FUNCTION_BLOCK SawmillMessageHandler
  (* Standard: 61499-2 *)
  (* Version 0.1, 2017-00-16, hpea485, UOA *)
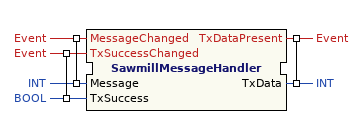
  EVENT_INPUT
    MessageChanged WITH Message;
    TxSuccessChanged WITH TxSuccess;
  END_EVENT
  EVENT_OUTPUT
    TxDataPresent WITH TxData;
  END_EVENT
  VAR_INPUT
    Message : INT;
    TxSuccess : BOOL;
  END_VAR
  VAR_OUTPUT
    TxData : INT;
  END_VAR
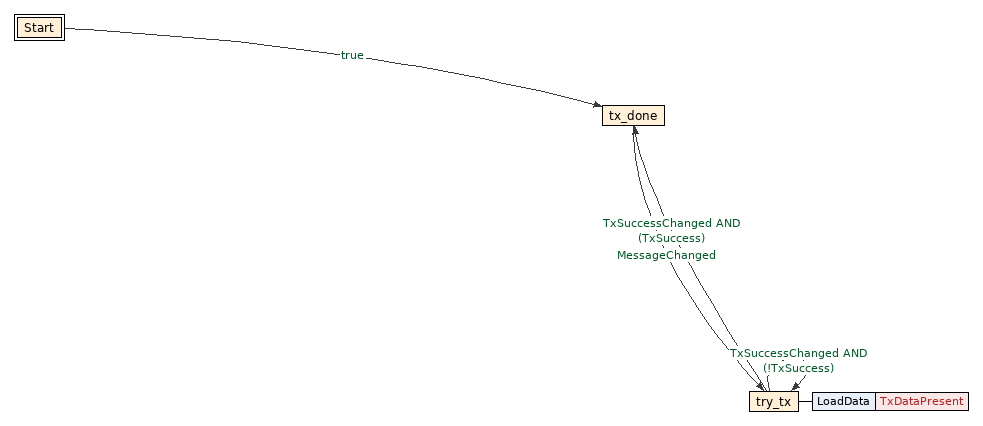
  EC_STATES
    Start;
    try_tx : LoadData -> TxDataPresent;
    tx_done;
  END_STATES
  EC_TRANSITIONS
    Start TO tx_done := true;
    try_tx TO try_tx := TxSuccessChanged AND (!TxSuccess);
    try_tx TO tx_done := TxSuccessChanged AND (TxSuccess);
    tx_done TO try_tx := MessageChanged;
  END_TRANSITIONS
  ALGORITHM LoadData IN C:
me->TxData = me->Message;
  END_ALGORITHM
END_FUNCTION_BLOCK
